PROGRAM MAIN
VAR
	bInit		: BOOL := TRUE;
	i			: INT;
	aDatos		: ARRAY[1..100] OF ST_Datos;
END_VAR

IF bInit THEN
	FOR i:=1 TO 100 DO
		aDatos[i].rValue1 := i*10.0;
		aDatos[i].nNumber := i;
	END_FOR
	bInit := FALSE;
END_IF

END_PROGRAM

(* stored: Version 1.1.0.1
   POU MAIN: Id {472135db-feb8-4ddf-83fe-fef2234cd41d}, SpecialFunc None *)
